// TIA Portal V20 export
TYPE "LER_typeJobInterface"
// stored: Access Published
   STRUCT
      motionRequest { ExternalWritable := 'False'} : Bool;
      loadingRequest { ExternalWritable := 'False'} : Bool;
      loadingReady { ExternalWritable := 'False'} : Bool;
      loadingDone { ExternalWritable := 'False'} : Bool;
      unLoadingRequest { ExternalWritable := 'False'} : Bool;
      unLoadingReady { ExternalWritable := 'False'} : Bool;
      unLoadingDone { ExternalWritable := 'False'} : Bool;
      clampRequest { ExternalWritable := 'False'} : Bool;
      clampReady { ExternalWritable := 'False'} : Bool;
      clampDone { ExternalWritable := 'False'} : Bool;
      unClampRequest { ExternalWritable := 'False'} : Bool;
      unClampReady { ExternalWritable := 'False'} : Bool;
      unClampDone { ExternalWritable := 'False'} : Bool;
      workingDone { ExternalWritable := 'False'} : Bool;
   END_STRUCT;
END_TYPE
